(* PLC project Template Project, Machine Expert Logic Builder V25.0.24.0, author Khaled HAMIDI *)
(* stored: creationDateTime 2026-08-29T10:46:10.3246713, version 0.0.0.1, modificationDateTime 2026-08-29T10:13:25.577481, organization Kur otomasyon *)

// TimeDate is not DateTime becouse its in usage.
TYPE TimeData :
STRUCT
    Act : SysTimeRtc.SYSTIMEDATE;   // -> HMI display
    Set : SysTimeRtc.SYSTIMEDATE;   // <- HMI edit fields
END_STRUCT
END_TYPE

TYPE MachineStatus :
STRUCT
    // ---- COMMAND : HMI writes ----
    Power       : BOOL;     // is power OK
    Home        : BOOL;     // is home
    ManualMode      : BOOL;     // NOT Auto
	AutoMode        : BOOL;     // auto / manual selector

	ResetRequest	:BOOL;	// true if reset requert
	StopRequest		:BOOL; 
    // ---- STATUS : PLC writes ----
    SafetyOk    : BOOL;     // emergency + doors
    BusOk       : BOOL;     // fieldbus ready
    PowerOk     : BOOL;     // all drives powered
    HomeOk      : BOOL;     // all axes homed
    AxisOk      : BOOL;     // all axes no error
    Ready       : BOOL;     // all above + no alarm

    Running     : BOOL;     // machine running
END_STRUCT
END_TYPE

(*
========================================
  HMI VARIABLE LIST
========================================

--- READ ---
Machine.Ready
Machine.Running
Machine.SafetyOk
Machine.PowerOk
Machine.HomeOk

Alarms.Active
Alarms.Count
Alarms.ActiveList[1..20]

Clock.Act.wDay
Clock.Act.wMonth
Clock.Act.wYear
Clock.Act.wHour
Clock.Act.wMinute
Clock.Act.wSecond


--- WRITE ---
Machine.Auto
Machine.Power
Machine.Home

Clock.Set.wDay
Clock.Set.wMonth
Clock.Set.wYear
Clock.Set.wHour
Clock.Set.wMinute
Clock.Set.wSecond

TimeRead        // button "Load"
TimeWrite       // button "Apply"


========================================
  TIME CHANGE
========================================
1. press "Load"     -> Clock.Set = Clock.Act
2. edit Clock.Set fields
3. press "Apply"    -> written to RTC

*)

TYPE hmi_table :
STRUCT
   
END_STRUCT
END_TYPE

PROGRAM SR_Main
VAR
END_VAR

                  DateTime();

Main._01_DefineButtons();
Main._02_DefineAlarms();
Main._03_MachineControl();
Main();

                
END_PROGRAM

FUNCTION_BLOCK Button

VAR_INPUT
    Signal : BOOL;        // Giriş sinyali
END_VAR

VAR_OUTPUT
    State      : BOOL;    // Anlık buton durumu
    Pressed    : BOOL;    // Basılma olayı (0 -> 1)
    Released  : BOOL;    // Bırakılma olayı (1 -> 0)
END_VAR

                  // Rising edge 0 -> 1
Pressed := Signal AND NOT State;

// Falling edge 1 -> 0
Released := NOT Signal AND State;

// Save Current state
State := Signal;
                
END_FUNCTION_BLOCK

FUNCTION_BLOCK Emergency

VAR_INPUT
    Signal : BOOL;
END_VAR

VAR_OUTPUT
    OK : BOOL;		// when signal equal to TRUE.
    Active: BOOL;	// = True when signal is FALSE
END_VAR

                  OK := Signal;
Active := NOT Ok;
                
END_FUNCTION_BLOCK

FUNCTION_BLOCK AlarmSystem
VAR_INPUT
    Reset       : BOOL;
END_VAR
VAR_OUTPUT
    Active      : BOOL;                         // -> HMI lamp
    Count       : UINT;                         // -> HMI
    ActiveList  : ARRAY [1..20] OF UINT;        // -> HMI list
END_VAR
VAR
    Cond        : ARRAY [1..100] OF BOOL;
    Latch       : ARRAY [1..100] OF BOOL;
    ResetTrig   : R_TRIG;
    BuzzerTon   : TON;
    BuzzerLtc   : BOOL;
    i           : UINT;
    idx         : UINT;
END_VAR

                  // CALL LAST, AFTER ALL Chk() CALLS

ResetTrig(CLK := Reset);

Count := 0;
idx   := 0;

FOR i := 1 TO 100 DO

    // reset clears only alarms whose condition is gone
    IF ResetTrig.Q AND NOT Cond[i] THEN
        Latch[i] := FALSE;
    END_IF

    IF Latch[i] THEN
        Count := Count + 1;
        IF idx < 20 THEN
            idx := idx + 1;
            ActiveList[idx] := i;
        END_IF
    END_IF

END_FOR

FOR i := idx + 1 TO 20 DO
    ActiveList[i] := 0;
END_FOR

Active := (Count > 0);

IF ResetTrig.Q THEN
    BuzzerLtc := FALSE;
END_IF

BuzzerTon(IN := BuzzerLtc, PT := T#5S);

IF BuzzerTon.Q THEN
    BuzzerLtc := FALSE;
END_IF
                

METHOD PUBLIC  Chk
VAR_INPUT
    ID      : UINT;
    Alarm   : BOOL;
END_VAR
                        IF (ID < 1) OR (ID > 100) THEN
    RETURN;
END_IF

Cond[ID] := Alarm;

IF Alarm AND NOT Latch[ID] THEN
    Latch[ID] := TRUE;
    BuzzerLtc := TRUE;
END_IF
                      
END_METHOD
END_FUNCTION_BLOCK

PROGRAM DateTime
VAR
    RTCget      : DWORD;
    SetTime     : DWORD;
    pRes        : SysTimeRtc.RTS_IEC_RESULT;
    TimeLoaded  : BOOL;
END_VAR

                  // ---------- READ RTC ----------
SysTimeRtc.SysTimeRtcConvertUtcToDate(dwTimestampUtc := RTCget, pDate := Clock.Act);
SysTimeRtc.SysTimeRtcGet(pResult := pRes, SysTimeRtcGet => RTCget);

// ---------- LOAD CURRENT TIME INTO EDIT FIELDS ----------
IF TimeRead THEN
    Clock.Set  := Clock.Act;
    TimeRead   := FALSE;
    TimeLoaded := TRUE;
END_IF

// ---------- WRITE RTC ----------
IF TimeWrite AND TimeLoaded THEN
    SysTimeRtc.SysTimeRtcConvertDateToUtc(pDate := Clock.Set, pdwTimestampUtc := SetTime);
    SysTimeRtc.SysTimeRtcSet(ulTimestamp := SetTime);
    TimeWrite  := FALSE;
    TimeLoaded := FALSE;
END_IF
                
END_PROGRAM

PROGRAM Main
VAR
	startButton		:	Button;
	stopButton		:	Button;
	reset		:	Emergency;
	emergencyStop	:	Emergency;
	
	
    // ---------- MASTER ----------
    MasterPower     : PLCO.MC_Power;
    MasterHome      : PLCO.MC_Home;
    MasterRun       : PLCO.MC_MoveVelocity;
    MasterStop      : PLCO.MC_Stop;

    // ---------- MOTOR 1 ----------
    M1Power         : PLCO.MC_Power;
    M1Home          : PLCO.MC_Home;
    M1Reset         : PLCO.MC_Reset;
    M1GearIn        : PLCO.MC_GearIn;
    M1Run           : PLCO.MC_MoveVelocity;
    M1Stop          : PLCO.MC_Stop;

    // ---------- MOTOR 2 ----------
    M2Power         : PLCO.MC_Power;
    M2Home          : PLCO.MC_Home;
    M2Reset         : PLCO.MC_Reset;
    M2GearIn        : PLCO.MC_GearIn;
	
	  // ---------- SETTINGS ----------
    Motor1Speed : LREAL := 50.0;    // deg/s   <- HMI
    Motor1Accel : LREAL := 200.0;
    Motor1Decel : LREAL := 200.0;

    // ---------- STATUS ----------
    Motor1Pos   : LREAL;            // -> HMI
END_VAR

                  // --------- CHECK StATUS -----
Machine.AxisOk		:= (DRV1.Axis.etAxisState <> 0);
Machine.BusOk		:= TRUE;
Machine.HomeOk		:= TRUE;
Machine.PowerOk		:= TRUE;
Machine.SafetyOk	:= TRUE;


///========= MOTORS =================
// ---------- RESET ----------
M1Reset( Axis    := DRV1.Axis,
         Execute := Machine.ResetRequest	);

// ---------- POWER ----------
M1Power( Axis   := DRV1.Axis,
         Enable := Machine.Power );

Machine.PowerOk := M1Power.Status;

// ---------- RUN ----------
M1Run( Axis         := DRV1.Axis,
       Execute      := Machine.Running,
       Velocity     := Motor1Speed,
       Acceleration := Motor1Accel,
       Deceleration := Motor1Decel );

// ---------- STOP ----------
M1Stop( Axis         := DRV1.Axis,
        Execute      := NOT Machine.Running,
        Deceleration := Motor1Decel );

// ---------- STATUS ----------
Motor1Pos := DRV1.Axis.lrPosition;

                

ACTION Run_Manual:
                      
                    
END_ACTION

ACTION _01_DefineButtons:
                      // Define Elements.

startButton(
	signal	:=	StartButton_In // start button OR from HMI or start button2 ... NO
);

stopButton(
	signal	:=	StopButton_In 	// stop button OR HMI or stop button2 ... NO
);

emergencyStop(
	Signal	:=	Emergency_In	// button1 AND button2 AND button3 NC
);

reset(
	signal := ResetButton_In	// from FSR .. normal Close NC.
);	

                    
END_ACTION

ACTION _02_DefineAlarms:
                      Alarms.Chk(  1, emergencyStop.Active          );  // Emergency Stop

// 100 .. System logic 

// 200 .. Sensors

// 400 .. > 499 Motors Drivers
Alarms.Chk( 41, (DRV1.Axis.etAxisState = 0)     );  // Motor 1 Fault

// ---- RUN  ----
Alarms( Reset := reset.Active );
                    
END_ACTION

ACTION _03_MachineControl:
                      Machine.Ready    := Machine.SafetyOk
                    AND Machine.BusOk
                    AND Machine.PowerOk
                    AND Machine.HomeOk
                    AND Machine.AxisOk
                    AND NOT Alarms.Active;

Machine.ResetRequest	:= Alarms.Active OR reset.Active;
// must be later in FB for machine status so its auto do this.. Machine.StopRequest		:= 
IF IS_DEBUG THEN
	Machine.Ready := TRUE;
	Machine.Running:= TRUE;
	
	AutoMode_Sw :=TRUE;
	
	StartButton_In :=TRUE;
	Emergency_In:= TRUE;
	StopButton_In :=FALSE;
	ResetButton_In :=TRUE;
END_IF

// ---------- MODE ----------
Machine.ManualMode := ManualMode_Sw;
Machine.AutoMode := AutoMode_Sw  AND NOT Machine.ManualMode;


// ---------- START / STOP ----------
IF StartButton.Pressed AND Machine.Ready AND (Machine.AutoMode OR Machine.ManualMode) THEN
    Machine.Running := TRUE;
END_IF

IF StopButton.Pressed OR NOT Machine.Ready THEN
    Machine.Running := FALSE;
END_IF

// ---------- Lamps ----------
AlarmLamp_Out 	:= Alarms.Active;
RunLamp_Out  	:= Machine.Running;
ReadyLamp_Out	:= Machine.Ready AND NOT Machine.Running;


// -------------- Call Methods -----------
IF Machine.AutoMode AND Machine.Running THEN
    Main.Run_Automatic();
END_IF

IF Machine.ManualMode AND Machine.Running THEN
    Main.Run_Manual();
END_IF

                    
END_ACTION

ACTION Run_Automatic:
                      
                    
END_ACTION
END_PROGRAM

CONFIGURATION Application
  RESOURCE Application ON PLC
(* global variable list GVL_IO *)
VAR_GLOBAL
	
    // ---------- DIGITAL INPUTS ----------
	(* Buttons *)
    StartButton_In      : BOOL;
    StopButton_In       : BOOL;
    ResetButton_In      : BOOL;
    Emergency_In        : BOOL;     // NC contact -> TRUE = OK
	
	(* Switchs *)
	ManualMode_Sw			: BOOL;
	AutoMode_Sw				: BOOL;			

    // ---------- DIGITAL OUTPUTS ----------
    (* Lamp *)
	RunLamp_Out       	: BOOL;
	ReadyLamp_Out		: BOOL;
    AlarmLamp_Out       : BOOL;


    // ---------- VIRTUAL MASTER ----------
    MasterAxis  : MOIN.FB_ControlledAxis;

    // ---------- REAL AXES ----------
    MainChain   : MOIN.FB_ControlledAxis;   // DRV1
    Conveyor    : MOIN.FB_ControlledAxis;   // DRV2
    CutterAxis  : MOIN.FB_ControlledAxis;   // DRV3

END_VAR
(* global variable list GVL_System *)
VAR_GLOBAL

    // ---------- ALARMS ----------
    Alarms      : AlarmSystem;

    // ---------- DATE / TIME ----------
    Clock       : TimeData;
    TimeRead    : BOOL;     // <- HMI button "Load"
    TimeWrite   : BOOL;     // <- HMI button "Apply"

	// --------- SYSTEM --------------
	Machine		: MachineStatus;
END_VAR
(* global variable list GVL_Recipe *)
VAR_GLOBAL
	
	IS_DEBUG: BOOL := TRUE;	
END_VAR
    TASK MAST(INTERVAL := T#10ms, PRIORITY := 15);
    PROGRAM SR_Main WITH MAST : SR_Main;
  END_RESOURCE
END_CONFIGURATION
